// TIA Portal project "lab5" (V15)

(* hardware
DEVICE "S7-1200 station_1"  S7-1200 Station
   slot 0: "Rack_0"  S7-1200 Rack  Rack  V1.0
   slot 1: "PLC_1"  CPU 1214C DC/DC/DC  6ES7 214-1AG40-0XB0  V4.1
      slot 3: "AI 1xRTD_1"  AI1 x RTD signal board  6ES7 231-5PA30-0XB0  V2.0
   slot 2: "AI 4x13BIT/AQ 2x14BIT_1"  6ES7 234-4HE32-0XB0  V2.0
*)

// ===== PLC "PLC_1"  CPU 1214C DC/DC/DC =====

VAR_GLOBAL   // PLC tag table "Default tag table"
   "MERENJE_TEMPERATURE_PT100" AT %IW80 : Int;   // 10 * T [Celsius]
   "UPRAVLJANJE_GREJACA" AT %QW96 : Int;   // 0 - 27700
   "ref" AT %MD100 : Real;
   "u_proc" AT %MD104 : Real;
   "auto_current" AT %M108.0 : Bool;
   "auto_previous" AT %M108.1 : Bool;
   "u_man" AT %MW109 : Word;
END_VAR

DATA_BLOCK "PI_REGULATOR_DB"   // DB1
{ S7_Optimized_Access := 'TRUE' }
VERSION : 0.1
// stored: InstanceOfName PI_REGULATOR
"PI_REGULATOR"
BEGIN
END_DATA_BLOCK

FUNCTION_BLOCK "PI_REGULATOR"   // FB1, SCL
{ S7_Optimized_Access := 'TRUE' }
VERSION : 0.1
   VAR_INPUT
      r : Real;
      y : Word;
      Kp : Real;
      Ti : Real;
      Ts : Real;
      u_man : Word;
   END_VAR
   VAR_OUTPUT
      u : Word;
      u_proc : Real;
   END_VAR
   VAR
      "e" : Real;
      up : Real;
      ui : Real;
      u_PI : Real;
      y_float : Real;
      u_man_float : Real;
   END_VAR
BEGIN
   // PI regulator - P (Proportional Gain), I (Integral Gain)

   // Na P (Proportional Gain) utice parametar Kp.
   // Sto je vece Kp, to sistem brze reaguje na gresku (razliku izmedju trenutne izmerene temperature i zeljene, tj.
   // reference -> e = r - y_float), tj. agresivnije ce da menja temperaturu.
   // Tada sistem brze postize zeljenu temperaturu, ali postoji rizik od "overshoot-a", tj da se zeljena temperatura
   // premasi, pa da je potrebno da se postepeno vrati temperatura na zeljenu, kada sistem ulazi u stacionarno stanje
   // kada temperatura oscilira oko zeljene.
   // Takodje, sto je vece Kp, to je veca verovatnoca da budu manje oscilacije nakon sto sistem udje u stacionarno
   // stanje, tj. veca je preciznost u stacionarnom stanju.

   // Na I (Integral Gain) utice parametar Ti.
   // Sto je vece Ti, to sistem blaze i postepenije ispravlja akumulirane greske iz proslosti kako bi se postiglo
   // sto preciznije stacionarno stanje, tj. da se odrzava temperatura sto blize zeljenoj.

   #y_float := #y / 10.0;
   #u_man_float := #u_man / 27700.0 * 100.0;

   IF "auto_current" THEN
       // Obezbedjivanje Bumpless prelaza izmedju rucnog i automatskog rezima rada.
       IF NOT "auto_previous" THEN
           #r := #y_float;
           #ui := #u_man_float;
       END_IF;
       #e := #r - #y_float;
       #up := #Kp * #e;
       #ui := #ui + #Kp / #Ti * #Ts * #e;
       #u_PI := #up + #ui;
       // Obezbedjivanje Antiwindup mehanizma u okviru automatskog rezima rada.
       IF #ui > 100.0 THEN
           #ui := 100.0;
       END_IF;
       IF #ui < 0.0 THEN
           #ui := 0.0;
       END_IF;
       IF #u_PI > 100.0 THEN
           #u_PI := 100.0;
       END_IF;
       IF #u_PI < 0.0 THEN
           #u_PI := 0.0;
       END_IF;
       #u_proc := #u_PI;
       #u := REAL_TO_INT(#u_PI / 100.0 * 27700.0);
       "auto_previous" := true;
   ELSE
       IF #u_man > 27700 THEN
           #u := 27700;
       ELSE
           IF #u_man < 0 THEN
               #u := 0;
           ELSE
               #u := #u_man;
           END_IF;
       END_IF;
       // Obezbedjivanje Bumpless prelaza izmedju rucnog i automatskog rezima rada.
       #r := #y_float;
       "auto_previous" := false;
   END_IF;
END_FUNCTION_BLOCK

ORGANIZATION_BLOCK "Main"   // OB1, LAD, ProgramCycle
TITLE = "Main Program Sweep (Cycle)"
{ S7_Optimized_Access := 'TRUE' }
VERSION : 0.1
   VAR_INPUT
      Initial_Call : Bool;   // Initial call of this OB
      Remanence : Bool;   // =True, if remanent data are available
   END_VAR
BEGIN
END_ORGANIZATION_BLOCK

ORGANIZATION_BLOCK "Cyclic interrupt"   // OB30, LAD, CyclicInterrupt
{ S7_Optimized_Access := 'TRUE' }
VERSION : 0.1
   VAR_INPUT
      Initial_Call : Bool;   // Initial call of this OB
      Event_Count : Int;   // Events discarded
   END_VAR
BEGIN

REGION Network 1
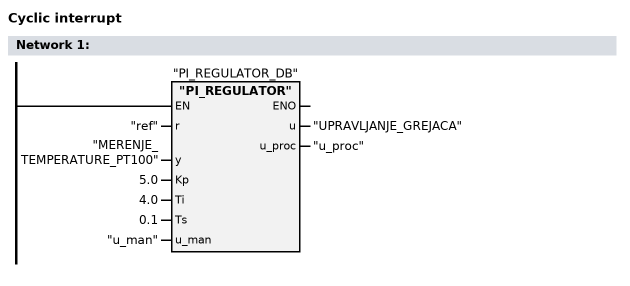
   RUNG wire#powerrail
      "PI_REGULATOR_DB"(r := "ref", y := "MERENJE_TEMPERATURE_PT100", Kp := 5.0, Ti := 4.0, Ts := 0.1, u_man := "u_man", u => "UPRAVLJANJE_GREJACA", u_proc => "u_proc")
   END_RUNG
   // the same network as SCL:
   "PI_REGULATOR_DB"(r := "ref",   // "PI_REGULATOR"
                     y := "MERENJE_TEMPERATURE_PT100",
                     Kp := 5.0,
                     Ti := 4.0,
                     Ts := 0.1,
                     u_man := "u_man",
                     u => "UPRAVLJANJE_GREJACA",
                     u_proc => "u_proc");
END_REGION
END_ORGANIZATION_BLOCK

ORGANIZATION_BLOCK "Startup"   // OB100, LAD, Startup
TITLE = "Complete Restart"
{ S7_Optimized_Access := 'TRUE' }
VERSION : 0.1
   VAR_INPUT
      LostRetentive : Bool;   // True if retentive data are lost
      LostRTC : Bool;   // True if date and time are lost
   END_VAR
BEGIN

REGION Network 1
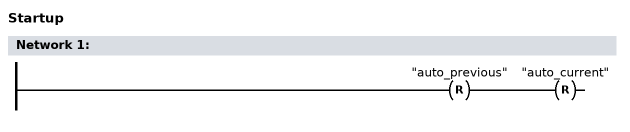
   RUNG wire#powerrail
      R_Coil( "auto_previous" )
      R_Coil( "auto_current" )
   END_RUNG
   // the same network as SCL:
   "auto_previous" := FALSE;
   "auto_current" := FALSE;
END_REGION
END_ORGANIZATION_BLOCK